% RSLogix 500 project Automatic Compressor with HOA.RSS, saved by version 8.30.00.16 %
PROJECT "UNTITLED"    % processor: Bul.1763 MicroLogix 1100 Series B %

PROGRAM FILES
  LAD 2 "MAIN"  7 rungs
  LAD 3 "INPUTS"  5 rungs
  LAD 4 "OUTPUTS"  3 rungs
  LAD 5 "CONTROLS"  10 rungs
  LAD 6 "ALARMS"  10 rungs

DATA FILES
  O0 OUTPUT  4 elements
  I1 INPUT  6 elements
  S2 STATUS  66 elements
  B3 BINARY  3 elements
  T4 TIMER  3 elements
  C5 COUNTER  1 elements
  R6 CONTROL  1 elements
  N7 INTEGER  2 elements
  F8 FLOAT  1 elements

LADDER 2 "MAIN"
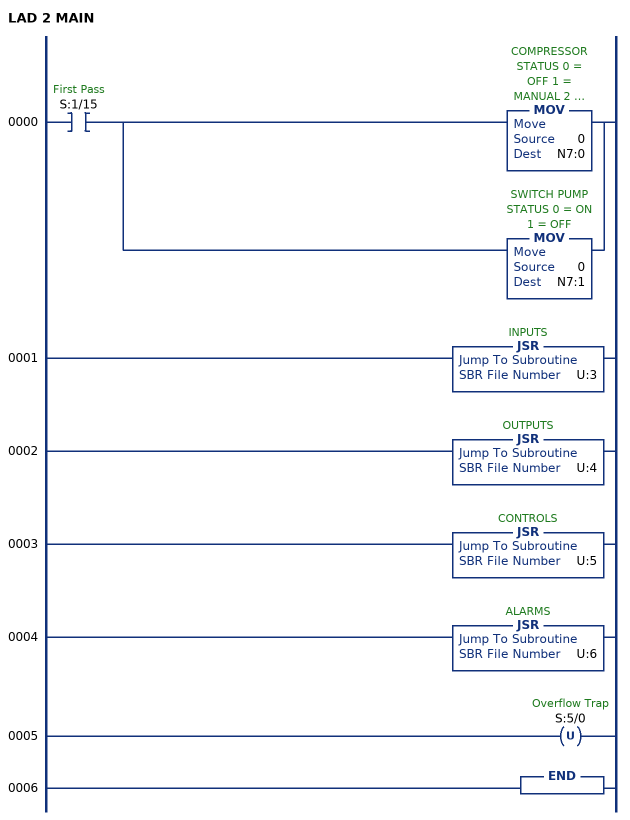
% Rung: 0 %
SOR XIC S:1/15 BST MOV 0 N7:0 NXB MOV 0 N7:1 BND EOR
%   S:1/15  "First Pass" %
%   N7:0  "COMPRESSOR STATUS 0 = OFF 1 = MANUAL 2 = AUTO" %
%   N7:1  "SWITCH PUMP STATUS 0 = ON 1 = OFF" %
% Rung: 1 %
SOR JSR U:3 EOR
%   U:3  "INPUTS" %
% Rung: 2 %
SOR JSR U:4 EOR
%   U:4  "OUTPUTS" %
% Rung: 3 %
SOR JSR U:5 EOR
%   U:5  "CONTROLS" %
% Rung: 4 %
SOR JSR U:6 EOR
%   U:6  "ALARMS" %
% Rung: 5 %
SOR OTU S:5/0 EOR
%   S:5/0  "Overflow Trap" %
% Rung: 6 %
SOR END EOR

LADDER 3 "INPUTS"
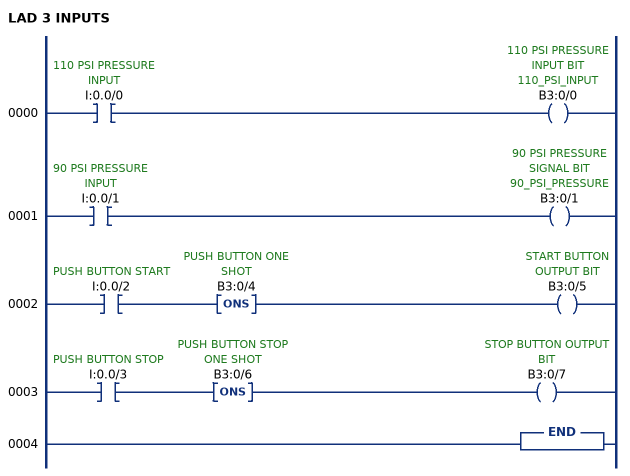
% Rung: 0 %
SOR XIC I:0.0/0 OTE B3:0/0 EOR
%   I:0.0/0  "110 PSI PRESSURE INPUT" %
%   B3:0/0  110_PSI_INPUT  "110 PSI PRESSURE INPUT BIT" %
% Rung: 1 %
SOR XIC I:0.0/1 OTE B3:0/1 EOR
%   I:0.0/1  "90 PSI PRESSURE INPUT" %
%   B3:0/1  90_PSI_PRESSURE  "90 PSI PRESSURE SIGNAL BIT" %
% Rung: 2 %
SOR XIC I:0.0/2 ONS B3:0/4 OTE B3:0/5 EOR
%   I:0.0/2  "PUSH BUTTON START" %
%   B3:0/4  "PUSH BUTTON ONE SHOT" %
%   B3:0/5  "START BUTTON OUTPUT BIT" %
% Rung: 3 %
SOR XIC I:0.0/3 ONS B3:0/6 OTE B3:0/7 EOR
%   I:0.0/3  "PUSH BUTTON STOP" %
%   B3:0/6  "PUSH BUTTON STOP ONE SHOT" %
%   B3:0/7  "STOP BUTTON OUTPUT BIT" %
% Rung: 4 %
SOR END EOR

LADDER 4 "OUTPUTS"
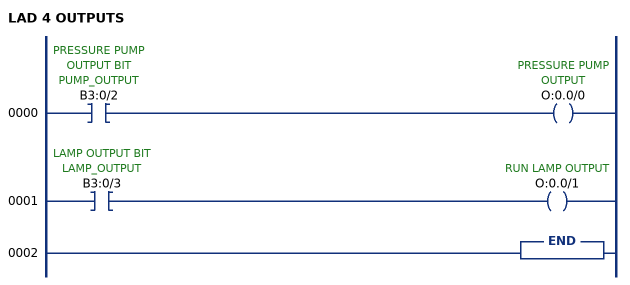
% Rung: 0 %
SOR XIC B3:0/2 OTE O:0.0/0 EOR
%   B3:0/2  PUMP_OUTPUT  "PRESSURE PUMP OUTPUT BIT" %
%   O:0.0/0  "PRESSURE PUMP OUTPUT" %
% Rung: 1 %
SOR XIC B3:0/3 OTE O:0.0/1 EOR
%   B3:0/3  LAMP_OUTPUT  "LAMP OUTPUT BIT" %
%   O:0.0/1  "RUN LAMP OUTPUT" %
% Rung: 2 %
SOR END EOR

LADDER 5 "CONTROLS"
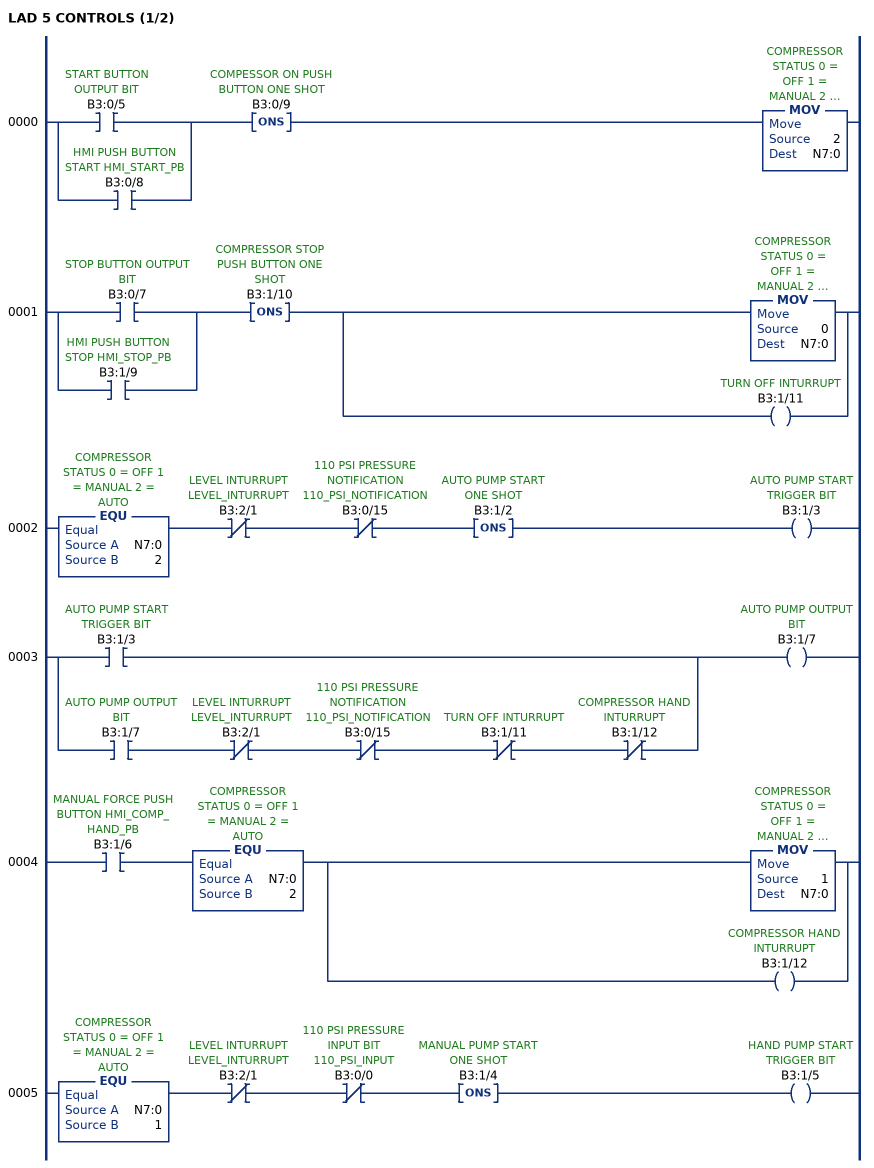
% Rung: 0 %
SOR BST XIC B3:0/5 NXB XIC B3:0/8 BND ONS B3:0/9 MOV 2 N7:0 EOR
%   B3:0/5  "START BUTTON OUTPUT BIT" %
%   B3:0/8  HMI_START_PB  "HMI PUSH BUTTON START" %
%   B3:0/9  "COMPESSOR ON PUSH BUTTON ONE SHOT" %
%   N7:0  "COMPRESSOR STATUS 0 = OFF 1 = MANUAL 2 = AUTO" %
% Rung: 1 %
SOR BST XIC B3:0/7 NXB XIC B3:1/9 BND ONS B3:1/10 BST MOV 0 N7:0 NXB OTE B3:1/11 BND EOR
%   B3:0/7  "STOP BUTTON OUTPUT BIT" %
%   B3:1/9  HMI_STOP_PB  "HMI PUSH BUTTON STOP" %
%   B3:1/10  "COMPRESSOR STOP PUSH BUTTON ONE SHOT" %
%   N7:0  "COMPRESSOR STATUS 0 = OFF 1 = MANUAL 2 = AUTO" %
%   B3:1/11  "TURN OFF INTURRUPT" %
% Rung: 2 %
SOR EQU N7:0 2 XIO B3:2/1 XIO B3:0/15 ONS B3:1/2 OTE B3:1/3 EOR
%   N7:0  "COMPRESSOR STATUS 0 = OFF 1 = MANUAL 2 = AUTO" %
%   B3:2/1  LEVEL_INTURRUPT  "LEVEL INTURRUPT" %
%   B3:0/15  110_PSI_NOTIFICATION  "110 PSI PRESSURE NOTIFICATION" %
%   B3:1/2  "AUTO PUMP START ONE SHOT" %
%   B3:1/3  "AUTO PUMP START TRIGGER BIT" %
% Rung: 3 %
SOR BST XIC B3:1/3 NXB XIC B3:1/7 XIO B3:2/1 XIO B3:0/15 XIO B3:1/11 XIO B3:1/12 BND OTE B3:1/7 EOR
%   B3:1/3  "AUTO PUMP START TRIGGER BIT" %
%   B3:1/7  "AUTO PUMP OUTPUT BIT" %
%   B3:2/1  LEVEL_INTURRUPT  "LEVEL INTURRUPT" %
%   B3:0/15  110_PSI_NOTIFICATION  "110 PSI PRESSURE NOTIFICATION" %
%   B3:1/11  "TURN OFF INTURRUPT" %
%   B3:1/12  "COMPRESSOR HAND INTURRUPT" %
% Rung: 4 %
SOR XIC B3:1/6 EQU N7:0 2 BST MOV 1 N7:0 NXB OTE B3:1/12 BND EOR
%   B3:1/6  HMI_COMP_HAND_PB  "MANUAL FORCE PUSH BUTTON" %
%   N7:0  "COMPRESSOR STATUS 0 = OFF 1 = MANUAL 2 = AUTO" %
%   B3:1/12  "COMPRESSOR HAND INTURRUPT" %
% Rung: 5 %
SOR EQU N7:0 1 XIO B3:2/1 XIO B3:0/0 ONS B3:1/4 OTE B3:1/5 EOR
%   N7:0  "COMPRESSOR STATUS 0 = OFF 1 = MANUAL 2 = AUTO" %
%   B3:2/1  LEVEL_INTURRUPT  "LEVEL INTURRUPT" %
%   B3:0/0  110_PSI_INPUT  "110 PSI PRESSURE INPUT BIT" %
%   B3:1/4  "MANUAL PUMP START ONE SHOT" %
%   B3:1/5  "HAND PUMP START TRIGGER BIT" %

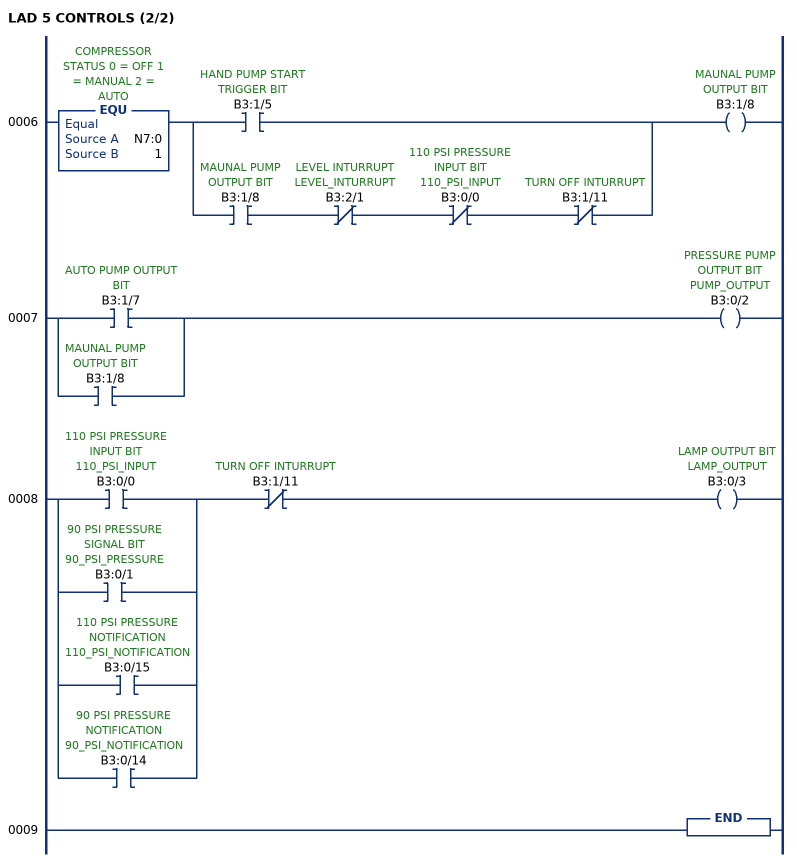
% Rung: 6 %
SOR EQU N7:0 1 BST XIC B3:1/5 NXB XIC B3:1/8 XIO B3:2/1 XIO B3:0/0 XIO B3:1/11 BND OTE B3:1/8 EOR
%   N7:0  "COMPRESSOR STATUS 0 = OFF 1 = MANUAL 2 = AUTO" %
%   B3:1/5  "HAND PUMP START TRIGGER BIT" %
%   B3:1/8  "MAUNAL PUMP OUTPUT BIT" %
%   B3:2/1  LEVEL_INTURRUPT  "LEVEL INTURRUPT" %
%   B3:0/0  110_PSI_INPUT  "110 PSI PRESSURE INPUT BIT" %
%   B3:1/11  "TURN OFF INTURRUPT" %
% Rung: 7 %
SOR BST XIC B3:1/7 NXB XIC B3:1/8 BND OTE B3:0/2 EOR
%   B3:1/7  "AUTO PUMP OUTPUT BIT" %
%   B3:1/8  "MAUNAL PUMP OUTPUT BIT" %
%   B3:0/2  PUMP_OUTPUT  "PRESSURE PUMP OUTPUT BIT" %
% Rung: 8 %
SOR BST XIC B3:0/0 NXB XIC B3:0/1 NXB XIC B3:0/15 NXB XIC B3:0/14 BND XIO B3:1/11 OTE B3:0/3 EOR
%   B3:0/0  110_PSI_INPUT  "110 PSI PRESSURE INPUT BIT" %
%   B3:0/1  90_PSI_PRESSURE  "90 PSI PRESSURE SIGNAL BIT" %
%   B3:0/15  110_PSI_NOTIFICATION  "110 PSI PRESSURE NOTIFICATION" %
%   B3:0/14  90_PSI_NOTIFICATION  "90 PSI PRESSURE NOTIFICATION" %
%   B3:1/11  "TURN OFF INTURRUPT" %
%   B3:0/3  LAMP_OUTPUT  "LAMP OUTPUT BIT" %
% Rung: 9 %
SOR END EOR

LADDER 6 "ALARMS"
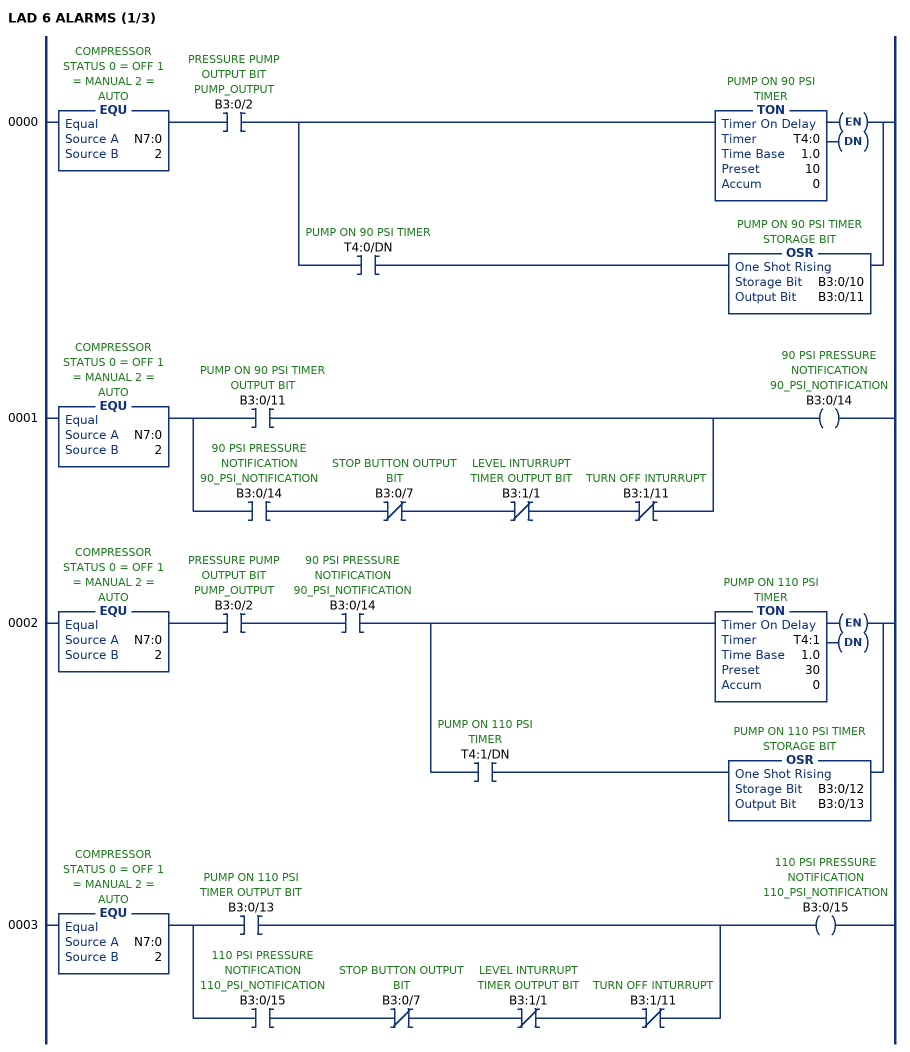
% Rung: 0 %
SOR EQU N7:0 2 XIC B3:0/2 BST TON T4:0 1.0 10 0 NXB XIC T4:0/DN OSR B3:0/10 B3:0/11 BND EOR
%   N7:0  "COMPRESSOR STATUS 0 = OFF 1 = MANUAL 2 = AUTO" %
%   B3:0/2  PUMP_OUTPUT  "PRESSURE PUMP OUTPUT BIT" %
%   T4:0  "PUMP ON 90 PSI TIMER" %
%   B3:0/10  "PUMP ON 90 PSI TIMER STORAGE BIT" %
%   B3:0/11  "PUMP ON 90 PSI TIMER OUTPUT BIT" %
% Rung: 1 %
SOR EQU N7:0 2 BST XIC B3:0/11 NXB XIC B3:0/14 XIO B3:0/7 XIO B3:1/1 XIO B3:1/11 BND OTE B3:0/14 EOR
%   N7:0  "COMPRESSOR STATUS 0 = OFF 1 = MANUAL 2 = AUTO" %
%   B3:0/11  "PUMP ON 90 PSI TIMER OUTPUT BIT" %
%   B3:0/14  90_PSI_NOTIFICATION  "90 PSI PRESSURE NOTIFICATION" %
%   B3:0/7  "STOP BUTTON OUTPUT BIT" %
%   B3:1/1  "LEVEL INTURRUPT TIMER OUTPUT BIT" %
%   B3:1/11  "TURN OFF INTURRUPT" %
% Rung: 2 %
SOR EQU N7:0 2 XIC B3:0/2 XIC B3:0/14 BST TON T4:1 1.0 30 0 NXB XIC T4:1/DN OSR B3:0/12 B3:0/13 BND EOR
%   N7:0  "COMPRESSOR STATUS 0 = OFF 1 = MANUAL 2 = AUTO" %
%   B3:0/2  PUMP_OUTPUT  "PRESSURE PUMP OUTPUT BIT" %
%   B3:0/14  90_PSI_NOTIFICATION  "90 PSI PRESSURE NOTIFICATION" %
%   T4:1  "PUMP ON 110 PSI TIMER" %
%   B3:0/12  "PUMP ON 110 PSI TIMER STORAGE BIT" %
%   B3:0/13  "PUMP ON 110 PSI TIMER OUTPUT BIT" %
% Rung: 3 %
SOR EQU N7:0 2 BST XIC B3:0/13 NXB XIC B3:0/15 XIO B3:0/7 XIO B3:1/1 XIO B3:1/11 BND OTE B3:0/15 EOR
%   N7:0  "COMPRESSOR STATUS 0 = OFF 1 = MANUAL 2 = AUTO" %
%   B3:0/13  "PUMP ON 110 PSI TIMER OUTPUT BIT" %
%   B3:0/15  110_PSI_NOTIFICATION  "110 PSI PRESSURE NOTIFICATION" %
%   B3:0/7  "STOP BUTTON OUTPUT BIT" %
%   B3:1/1  "LEVEL INTURRUPT TIMER OUTPUT BIT" %
%   B3:1/11  "TURN OFF INTURRUPT" %

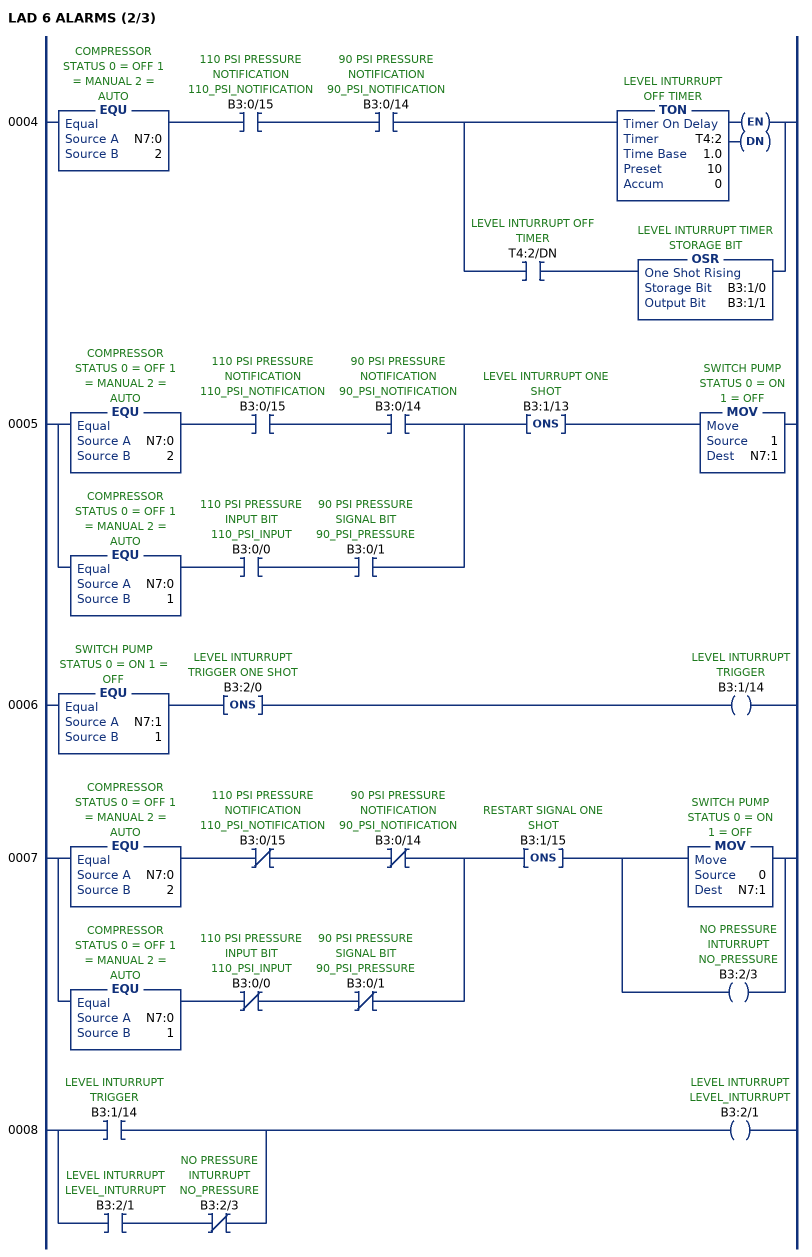
% Rung: 4 %
SOR EQU N7:0 2 XIC B3:0/15 XIC B3:0/14 BST TON T4:2 1.0 10 0 NXB XIC T4:2/DN OSR B3:1/0 B3:1/1 BND EOR
%   N7:0  "COMPRESSOR STATUS 0 = OFF 1 = MANUAL 2 = AUTO" %
%   B3:0/15  110_PSI_NOTIFICATION  "110 PSI PRESSURE NOTIFICATION" %
%   B3:0/14  90_PSI_NOTIFICATION  "90 PSI PRESSURE NOTIFICATION" %
%   T4:2  "LEVEL INTURRUPT OFF TIMER" %
%   B3:1/0  "LEVEL INTURRUPT TIMER STORAGE BIT" %
%   B3:1/1  "LEVEL INTURRUPT TIMER OUTPUT BIT" %
% Rung: 5 %
SOR BST EQU N7:0 2 XIC B3:0/15 XIC B3:0/14 NXB EQU N7:0 1 XIC B3:0/0 XIC B3:0/1 BND ONS B3:1/13 MOV 1 N7:1 EOR
%   N7:0  "COMPRESSOR STATUS 0 = OFF 1 = MANUAL 2 = AUTO" %
%   B3:0/15  110_PSI_NOTIFICATION  "110 PSI PRESSURE NOTIFICATION" %
%   B3:0/14  90_PSI_NOTIFICATION  "90 PSI PRESSURE NOTIFICATION" %
%   B3:0/0  110_PSI_INPUT  "110 PSI PRESSURE INPUT BIT" %
%   B3:0/1  90_PSI_PRESSURE  "90 PSI PRESSURE SIGNAL BIT" %
%   B3:1/13  "LEVEL INTURRUPT ONE SHOT" %
%   N7:1  "SWITCH PUMP STATUS 0 = ON 1 = OFF" %
% Rung: 6 %
SOR EQU N7:1 1 ONS B3:2/0 OTE B3:1/14 EOR
%   N7:1  "SWITCH PUMP STATUS 0 = ON 1 = OFF" %
%   B3:2/0  "LEVEL INTURRUPT TRIGGER ONE SHOT" %
%   B3:1/14  "LEVEL INTURRUPT TRIGGER" %
% Rung: 7 %
SOR BST EQU N7:0 2 XIO B3:0/15 XIO B3:0/14 NXB EQU N7:0 1 XIO B3:0/0 XIO B3:0/1 BND ONS B3:1/15 BST MOV 0 N7:1 NXB OTE B3:2/3 BND EOR
%   N7:0  "COMPRESSOR STATUS 0 = OFF 1 = MANUAL 2 = AUTO" %
%   B3:0/15  110_PSI_NOTIFICATION  "110 PSI PRESSURE NOTIFICATION" %
%   B3:0/14  90_PSI_NOTIFICATION  "90 PSI PRESSURE NOTIFICATION" %
%   B3:0/0  110_PSI_INPUT  "110 PSI PRESSURE INPUT BIT" %
%   B3:0/1  90_PSI_PRESSURE  "90 PSI PRESSURE SIGNAL BIT" %
%   B3:1/15  "RESTART SIGNAL ONE SHOT" %
%   N7:1  "SWITCH PUMP STATUS 0 = ON 1 = OFF" %
%   B3:2/3  NO_PRESSURE  "NO PRESSURE INTURRUPT" %
% Rung: 8 %
SOR BST XIC B3:1/14 NXB XIC B3:2/1 XIO B3:2/3 BND OTE B3:2/1 EOR
%   B3:1/14  "LEVEL INTURRUPT TRIGGER" %
%   B3:2/1  LEVEL_INTURRUPT  "LEVEL INTURRUPT" %
%   B3:2/3  NO_PRESSURE  "NO PRESSURE INTURRUPT" %

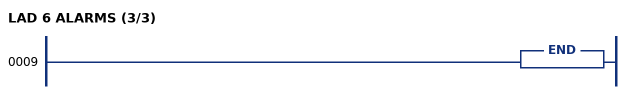
% Rung: 9 %
SOR END EOR

DATA TABLE (non-zero values as saved)
DATA T4
% .PRE .ACC %
% T4:0 % 10 0
% T4:1 % 30 0
% T4:2 % 10 0
